Universal Robots PolyScope program: xmlrpc_example_listadinamica_OK.urp

Program xmlrpc_example (installation=default directory=/home/ur/ursim-current/programs createdIn=5.17.0 lastSavedIn=5.17.0 robotSerialNumber=20195299999)
Calibrated DH parameters: a=[0, -0.6127, -0.57155, 0, 0, 0]; d=[0.1807, 0, 0, 0.17415, 0.11985, 0.11655]; alpha=[1.570796, 0, 0, 1.570796, -1.570796, 0]; deltaTheta=[0, 0, 0, 0, 0, 0]
InitVariablesNode
BeforeStart
  camera := rpc_factory("xmlrpc","http://192.168.56.250:50000")
Robot Program (runOnlyOnce=false)
  Loop While (checkContinuously=false) expression=True
    next_pose := camera.get_next_pose()
    If next_pose[0] == 0  and next_pose[1] == 0  and next_pose[2] == 0  and next_pose[3] == 0  and next_pose[4] ==0  and next_pose[5] == 0
      MoveJ speed 60 deg/s, acceleration 80 deg/s^2 (useActiveTCP=true) feature=Base
        Waypoint Casa: TCP in base x=-135.367 y=-436.496 z=231.741 mm, rx=1.2732 ry=2.5806 rz=-0.3859 rad; joints [-85.944, -88.585, -151.1, -10.245, 94.057, 57.296] deg
        Wait Sleep waitTime=1
    Else 
      MoveJ speed 60 deg/s, acceleration 80 deg/s^2 (useActiveTCP=true) feature=Base
        Waypoint Variable (Variable): variable=next_pose
    Script: sync()
